Fanuc TP program (LS listing): UP101.LS

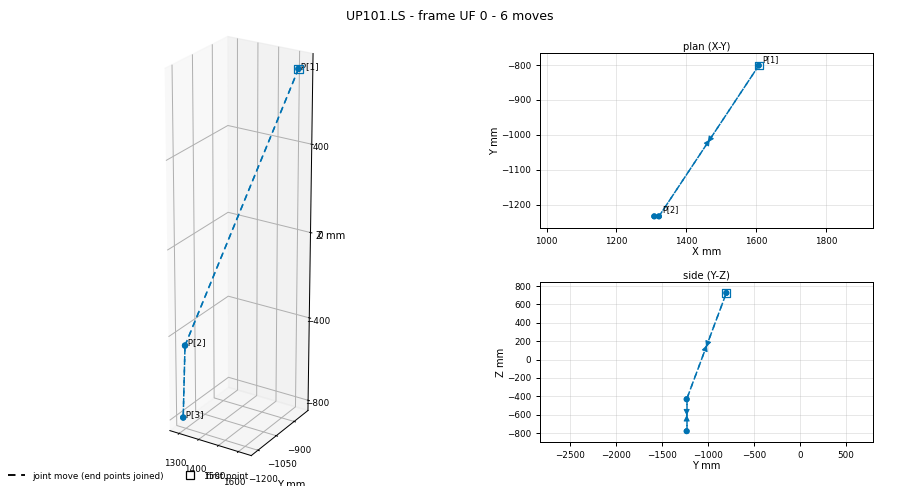
[picture p0: tool path of UP101.LS in frame UF 0, 6 of 7 moves have a stored position in this frame; points joined in program order, loops and branches not executed]
/PROG  UP101
/ATTR
OWNER		= AUROM;
COMMENT		= "Fresado";
PROG_SIZE	= 3868;
CREATE		= DATE 96-06-02  TIME 16:08:02;
MODIFIED	= DATE 23-08-22  TIME 15:31:38;
FILE_NAME	= UP101;
VERSION		= 0;
LINE_COUNT	= 14;
MEMORY_SIZE	= 6632;
PROTECT		= READ_WRITE;
TCD:  STACK_SIZE	= 500,
      TASK_PRIORITY	= 50,
      TIME_SLICE	= 0,
      BUSY_LAMP_OFF	= 0,
      ABORT_REQUEST	= 0,
      PAUSE_REQUEST	= 0;
DEFAULT_GROUP	= 1,1,1,1,*;
CONTROL_CODE	= 00000000 00000000;
/APPL
/MN
    :  UFRAME_NUM=0 ;
    :  UTOOL_NUM=1 ;
    :  PAYLOAD[1] ;
    :J P[1] 100% CNT0 ACC100 TB    .10sec,P-SPS    ;
      1:  TC_ONLINE (ON) ;
      2:  DO[23]=OFF ;
      3:  CALL MAKRO050    ;
      4:  !Lib. de Herramientas ;
      5:  DO[80]=ON ;
      6:  DO[79]=ON ;
      7:  !Lib. de Anticolisiones ;
      8:  DO[41]=ON ;
      9:  DO[42]=ON ;
     10:  DO[43]=ON ;
     11:  DO[44]=ON ;
     12:  !Apagar Pos. Base ;
     13:  DO[15]=OFF ;
     14:  !Robot en Trayectoria ;
     15:  DO[16]=ON ;
     16:  DO[756]=OFF ;
     17:  !Ap. Med. Ant/Dsp. Fresar ;
     18:  DO[756]=OFF ;
     19:  DO[757]=OFF ;
     20:  CALL VW_USER(Basic1,EZSP,Nr1 Service,ProgNr=31, , ,S-Punkt=31, ,EIN/AUS=1) ;
     21:  WAIT    .10(sec) ;
     22:  !Fresado Ciclico ;
     23:  F[79]=((DI[786] AND !DI[788]) OR F[298] OR (!DI[786] AND !DI[788] AND DO[11]) OR (!DI[788] AND DI[130])) ;
     24:  !Fresado Inicial ;
     25:  F[78]=(DI[788] AND !F[79]) ;
     26:  WAIT (DI[23])    ;
     27:  DO[23]=ON ;
     28:  TC_ONLINE (M[30] AND M[95]) ;
       ------ ;
    :J P[2] 100% CNT100 ACC100 TB   0.00sec,P-SPS    ;
      1:  TC_ONLINE (M[30] AND M[95]) ;
       ------ ;
    :J P[3] 100% CNT0 ACC100 TB    .10sec,P-SPS    ;
      1:  TC_ONLINE (ON) ;
      2:  DO[23]=OFF ;
      3:  WAIT (DI[23])    ;
      4:  DO[23]=ON ;
      5:  TC_ONLINE (M[30] AND M[95]) ;
       ------ ;
    :  !Pos. de Fresado ;
    :J P[4] 100% CNT0 ACC100 TB    .10sec,P-SPS Tool_Offset,PR[11] Offset,PR[12]    ;
      1:  TC_ONLINE (ON) ;
      2:  DO[23]=OFF ;
      3:  CALL VW_USER(Basic1,EZSP,Nr1 Service,ProgNr=31, , ,S-Punkt=31, ,EIN/AUS=1) ;
      4:  !Sel. de Pistola ;
      5:  F[64]=(ON) ;
      6:  F[65]=(OFF) ;
      7:  F[66]=(OFF) ;
      8:  F[67]=(OFF) ;
      9:  DO[130]=ON ;
     10:  GO[2]=(R[197]+5) ;
     11:  IF (F[78] OR F[79]),CALL MAKRO082 ;
     12:  DO[130]=OFF ;
     13:  WAIT (DI[23])    ;
     14:  DO[23]=ON ;
     15:  TC_ONLINE (M[30] AND M[95]) ;
       ------ ;
    :J P[5] 100% CNT0 ACC100 TB    .10sec,P-SPS    ;
      1:  TC_ONLINE (ON) ;
      2:  DO[23]=OFF ;
      3:  WAIT (DI[23])    ;
      4:  DO[23]=ON ;
      5:  TC_ONLINE (M[30] AND M[95]) ;
       ------ ;
    :  !Inic. de Med. ;
    :J P[6] 100% CNT100 ACC100 TB   0.00sec,P-SPS    ;
      1:  TC_ONLINE (ON) ;
      2:  DO[715]=ON ;
      3:  DO[757]=ON ;
      4:  TC_ONLINE (M[30] AND M[95]) ;
       ------ ;
    :  !Fin de Med. ;
    :  !Posicion Base ;
    :J P[7] 100% CNT0 ACC100 TB    .10sec,P-SPS    ;
      1:  TC_ONLINE (ON) ;
      2:  DO[23]=OFF ;
      3:  CALL MAKRO083    ;
      4:  IF (F[78] AND !F[79] AND F[335]),CALL MAKRO087 ;
      5:  CALL VW_USER(Basic1,EZSP,Nr1 Service,ProgNr=41, , ,S-Punkt=41, ,EIN/AUS=F[78]) ;
      6:  CALL VW_USER(Basic1,EZSP,Nr1 Service,ProgNr=51, , ,S-Punkt=51, ,EIN/AUS=F[79]) ;
      7:  IF (!F[85] AND !F[86]),CALL MAKRO080 ;
      8:  WAIT (!F[298] OR (DI[777] AND F[298]) OR DI[26] OR (F[298] AND F[749]))    ;
      9:  WAIT (DI[23])    ;
     10:  DO[23]=ON ;
     11:  TC_ONLINE (M[30] AND M[95]) ;
       ------ ;
/POS
P[1]{
   GP1:
	UF : 0, UT : 1,		CONFIG : 'N U T, 0, 0, 0',
	X =  1607.403  mm,	Y =  -801.498  mm,	Z =   725.794  mm,
	W =   176.848 deg,	P =   -29.910 deg,	R =   -22.694 deg
   GP2:
	UF : 0, UT : 1,
	J1=   100.000  mm
   GP3:
	UF : 0, UT : 1,
	J1=     0.000  mm
   GP4:
	UF : 0, UT : 1,
	J1=     0.000  mm
};
P[2]{
   GP1:
	UF : 0, UT : 1,		CONFIG : 'N U T, 0, 0, 0',
	X =  1321.560  mm,	Y = -1233.419  mm,	Z =  -431.887  mm,
	W =  -180.000 deg,	P =    -1.266 deg,	R =     0.000 deg
   GP2:
	UF : 0, UT : 1,
	J1=   100.000  mm
   GP3:
	UF : 0, UT : 1,
	J1=     0.000  mm
   GP4:
	UF : 0, UT : 1,
	J1=     0.000  mm
};
P[3]{
   GP1:
	UF : 0, UT : 1,		CONFIG : 'N U T, 0, 0, 0',
	X =  1308.125  mm,	Y = -1233.419  mm,	Z =  -779.909  mm,
	W =  -180.000 deg,	P =    -1.266 deg,	R =     0.000 deg
   GP2:
	UF : 0, UT : 1,
	J1=   100.000  mm
   GP3:
	UF : 0, UT : 1,
	J1=     0.000  mm
   GP4:
	UF : 0, UT : 1,
	J1=     0.000  mm
};
P[4]{
   GP1:
	UF : 0, UT : 1,		CONFIG : 'N U T, 0, 0, 0',
	X =  1377.711  mm,	Y = -1233.419  mm,	Z =  -777.610  mm,
	W =   180.000 deg,	P =    -1.266 deg,	R =      .000 deg
   GP2:
	UF : 0, UT : 1,
	J1=   100.000  mm
   GP3:
	UF : 0, UT : 1,
	J1=     0.000  mm
   GP4:
	UF : 0, UT : 1,
	J1=     0.000  mm
};
P[5]{
   GP1:
	UF : 0, UT : 1,		CONFIG : 'N U T, 0, 0, 0',
	X =  1308.125  mm,	Y = -1233.419  mm,	Z =  -779.909  mm,
	W =  -180.000 deg,	P =    -1.266 deg,	R =     0.000 deg
   GP2:
	UF : 0, UT : 1,
	J1=   100.000  mm
   GP3:
	UF : 0, UT : 1,
	J1=     0.000  mm
   GP4:
	UF : 0, UT : 1,
	J1=     0.000  mm
};
P[6]{
   GP1:
	UF : 0, UT : 1,		CONFIG : 'N U T, 0, 0, 0',
	X =  1321.560  mm,	Y = -1233.419  mm,	Z =  -431.887  mm,
	W =  -180.000 deg,	P =    -1.266 deg,	R =     0.000 deg
   GP2:
	UF : 0, UT : 1,
	J1=   100.000  mm
   GP3:
	UF : 0, UT : 1,
	J1=     0.000  mm
   GP4:
	UF : 0, UT : 1,
	J1=     0.000  mm
};
P[7]{
   GP1:
	UF : 0, UT : 1,		CONFIG : 'N U T, 0, 0, 0',
	X =  1607.403  mm,	Y =  -801.498  mm,	Z =   725.794  mm,
	W =   176.848 deg,	P =   -29.910 deg,	R =   -22.694 deg
   GP2:
	UF : 0, UT : 1,
	J1=   100.000  mm
   GP3:
	UF : 0, UT : 1,
	J1=     0.000  mm
   GP4:
	UF : 0, UT : 1,
	J1=     0.000  mm
};
/END
